// TIA Portal V19 export
ORGANIZATION_BLOCK "Main"   // OB1, LAD, ProgramCycle
TITLE = "Main Program Sweep (Cycle)"
{ S7_Optimized_Access := 'TRUE' }
// TIA Demo Project
// 1500 password is Siemens1
// stored: SetENOAutomatically false
   VAR_INPUT
      Initial_Call : Bool;   // Initial call of this OB
      Remanence : Bool;   // =True, if remanent data are available
   END_VAR
   VAR_TEMP   // added for the SCL form of the ladder/FBD networks
      _w1 : Bool;
      _w2 : Bool;
   END_VAR
BEGIN

REGION Network 1: Scale the Potentiometer raw value to a Real between 0.0-1500.0
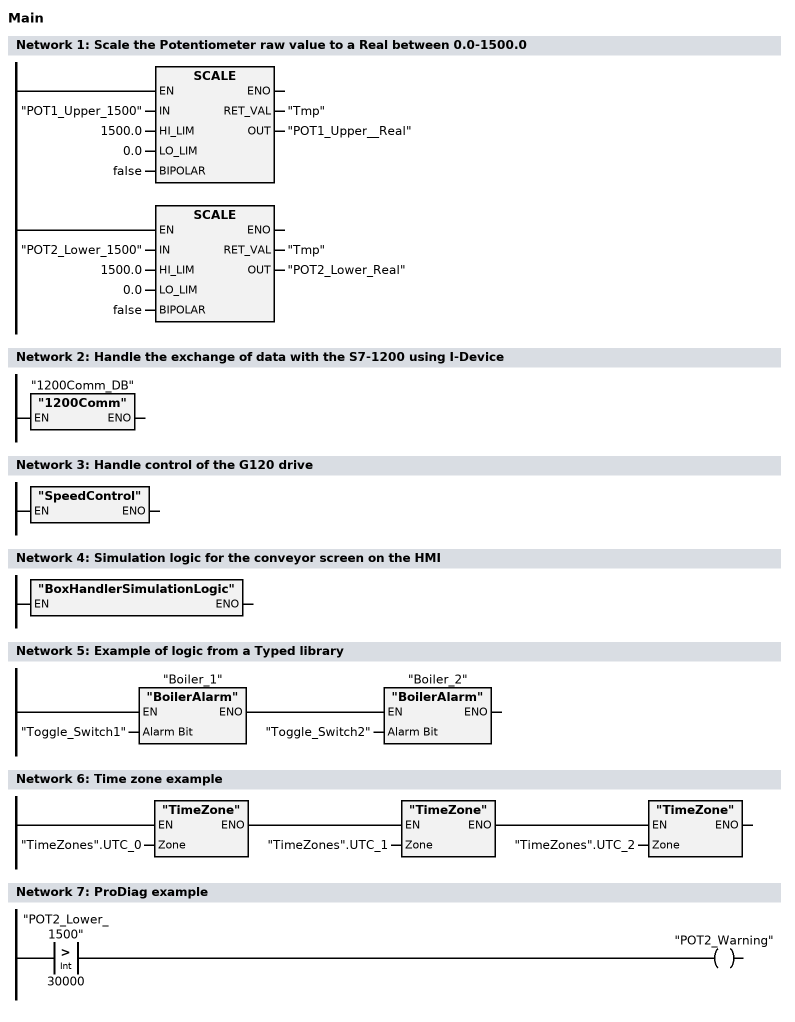
   "Tmp" := SCALE(IN := "POT1_Upper_1500",
                  HI_LIM := 1500.0,
                  LO_LIM := 0.0,
                  BIPOLAR := false,
                  OUT => "POT1_Upper__Real");
   "Tmp" := SCALE(IN := "POT2_Lower_1500",
                  HI_LIM := 1500.0,
                  LO_LIM := 0.0,
                  BIPOLAR := false,
                  OUT => "POT2_Lower_Real");
END_REGION

REGION Network 2: Handle the exchange of data with the S7-1200 using I-Device
   RUNG wire#powerrail
      "1200Comm_DB"()
   END_RUNG
   // the same network as SCL:
   "1200Comm_DB"();   // "1200Comm"
END_REGION

REGION Network 3: Handle control of the G120 drive
   RUNG wire#powerrail
      "SpeedControl"()
   END_RUNG
   // the same network as SCL:
   "SpeedControl"();
END_REGION

REGION Network 4: Simulation logic for the conveyor screen on the HMI
   RUNG wire#powerrail
      "BoxHandlerSimulationLogic"()
   END_RUNG
   // the same network as SCL:
   "BoxHandlerSimulationLogic"();
END_REGION

REGION Network 5: Example of logic from a Typed library
   RUNG wire#powerrail
      "Boiler_1"("Alarm Bit" := "Toggle_Switch1")
      "Boiler_2"("Alarm Bit" := "Toggle_Switch2")
   END_RUNG
   // the same network as SCL:
   "Boiler_1"("Alarm Bit" := "Toggle_Switch1", ENO => #_w1);   // "BoilerAlarm"
   IF #_w1 THEN
       "Boiler_2"("Alarm Bit" := "Toggle_Switch2");   // "BoilerAlarm"
   END_IF;
END_REGION

REGION Network 6: Time zone example
   RUNG wire#powerrail
      "TimeZone"(Zone := "TimeZones".UTC_0)
      "TimeZone"(Zone := "TimeZones".UTC_1)
      "TimeZone"(Zone := "TimeZones".UTC_2)
   END_RUNG
   // the same network as SCL:
   "TimeZone"(Zone := "TimeZones".UTC_0, ENO => #_w1);
   "TimeZone"(EN := #_w1, Zone := "TimeZones".UTC_1, ENO => #_w2);
   IF #_w2 THEN "TimeZone"(Zone := "TimeZones".UTC_2); END_IF;
END_REGION

REGION Network 7: ProDiag example
   RUNG wire#powerrail
      { S7_Templates := "SrcType := Int" } GT_Contact(in1 := "POT2_Lower_1500", in2 := 30000)
      Coil( "POT2_Warning" )
   END_RUNG
   // the same network as SCL:
   "POT2_Warning" := "POT2_Lower_1500" > 30000;
END_REGION
END_ORGANIZATION_BLOCK
